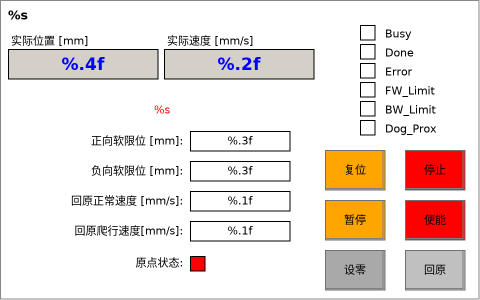
VISUALIZATION motionModuleP2  // 480x300
VAR_IN_OUT
	userData: motionModuleDataHMI;
END_VAR
    Rectangle (36,126 150x30), "正向软限位 [mm]:"
    Rectangle (190,131 100x20), "%.3f", text variable: userData.softPLimitPos, input disabled if: TRUE
        OnMouseDown: write the text variable via Edit
    Rectangle (36,156 150x30), "负向软限位 [mm]:"
    Rectangle (190,161 100x20), "%.3f", text variable: userData.softNLimitPos, input disabled if: TRUE
        OnMouseDown: write the text variable via Edit
    Rectangle (190,191 100x20), "%.1f", text variable: userData.goHomeVel
        OnMouseDown: write the text variable via Edit
    Button (405,250 60x40), "回原", colour toggle: userData.goHomeDone, input disabled if: NOT userData.homeCondition OR NOT userData.ctrlModeCondition
        tap userData.goHomeGo
    Rectangle (190,221 100x20), "%.1f", text variable: userData.goHomeVelSlow
        OnMouseDown: write the text variable via Edit
    Rectangle (36,186 150x30), "回原正常速度 [mm/s]:"
    Rectangle (27,216 159x30), "回原爬行速度[mm/s]:"
    Rectangle (79,248 107x30), "原点状态:"
    Rectangle (8,49 150x30), "%.4f", text variable: userData.actualPos
    Rectangle (8,26 150x30), "实际位置 [mm]"
    Rectangle (164,49 150x30), "%.2f", text variable: userData.actualVel
    Rectangle (164,26 150x30), "实际速度 [mm/s]"
    Rectangle (360,82 15x15), colour toggle: userData.forwardLimitSwitch
    Rectangle (360,101 15x15), colour toggle: userData.backwardsLimitSwitch
    Rectangle (360,120 15x15), colour toggle: userData.dogPointSwitch
    Rectangle (382,80 64x22), "FW_Limit"
    Rectangle (382,99 64x22), "BW_Limit"
    Rectangle (382,118 64x22), "Dog_Prox"
    Button (405,200 60x40), "使能", colour toggle: userData.powerEnable, input disabled if: NOT userData.ctrlModeCondition
        tap userData.power
    Button (325,250 60x40), "设零", invisible if: TRUE, input disabled if: NOT userData.setCondition OR NOT userData.ctrlModeCondition
        tap userData.setZero
    Button (325,200 60x40), "暂停", colour toggle: userData.oPause, input disabled if: NOT userData.ctrlModeCondition
        tap userData.pauseB
    Rectangle (190,256 15x15), colour toggle: userData.goHomeDone
    Rectangle (12,100 300x20), "%s", text variable: userData.errTxt
    Rectangle (5,5 467x20), "%s", text variable: userData.nameTXT
    Button (405,150 60x40), "停止"
        tap userData.stop
    Button (325,150 60x40), "复位"
        tap userData.reset
    Rectangle (360,25 15x15), colour toggle: userData.busy
    Rectangle (382,23 64x22), "Busy"
    Rectangle (382,42 64x22), "Done"
    Rectangle (382,61 64x22), "Error"
    Rectangle (360,44 15x15), colour toggle: userData.done
    Rectangle (360,63 15x15), colour toggle: userData.error
END_VISUALIZATION

(* stored: Version 1.1.0.1, ProductVersion 3.1.4024.4
   Visu motionModuleP2: Id {ef1bd2fb-8d4c-4ccb-9198-4ada169f471d} *)
